FUNCTION_BLOCK Cubic_Polynomial_Interpolation
//VAR_INPUT
//	t0,t1,q0,q1,v0,v1,acc0,acc1:LREAL;	
//	t:LREAL;
//END_VAR
VAR
	h,Tp:LREAL;
	a0,a1,a2,a3:LREAL;
	targetPos,targetVel,targetAcc:LREAL;
END_VAR



//IF (t<=t1) THEN
//	pos:=a0+a1*t+a2*EXPT(t,2)+a3*EXPT(t,3);
//	vel:=a1+2*a2*t+3*a3*EXPT(t,2);
//	acc:=2*a2+6*a3*t;
//END_IF

//IF (t>t1) THEN
//	finished:=TRUE;
//	pos:=q1;
//	vel:=0;
//	acc:=0;
//ELSE
//	finished:=FALSE;
//END_IF

METHOD init : BOOL
VAR_INPUT
	t0,t1,q0,q1,v0,v1,acc0,acc1:LREAL;	
END_VAR
targetPos:=0;
targetVel:=0;
targetAcc:=0;
a0:=0;
a1:=0;
a2:=0;
a3:=0;
h:=q1-q0;
Tp:=t1-t0;

a0:=q0;
a1:=v0;
a2:=3/EXPT(Tp,2)*h-2/Tp*v0-1/Tp*v1;
a3:=-2/EXPT(Tp,3)*h+1/EXPT(Tp,2)*(v1+v0);

targetPos:=q1;
targetVel:=v1;
targetAcc:=a1;
END_METHOD

METHOD run : BOOL
VAR_INPUT
	t:LREAL;
END_VAR
VAR_IN_OUT
	pos:lreal;
	vel:lreal;
	acc:LREAL;
END_VAR
IF t>Tp THEN
	pos:=targetPos;
	vel:=targetVel;
	acc:=targetAcc;
ELSE	
	pos:=a0+a1*t+a2*EXPT(t,2)+a3*EXPT(t,3);
	vel:=a1+2*a2*t+3*a3*EXPT(t,2);
	acc:=2*a2+6*a3*t;
END_IF
END_METHOD

END_FUNCTION_BLOCK

(* stored: Version 1.1.0.1, ProductVersion 3.1.4024.12
   POU Cubic_Polynomial_Interpolation: Id {d05795ca-46ae-45d1-a565-0dbdff11dcfb}, SpecialFunc None
   Method init: Id {b4cf89e5-ebd6-4df0-a5ad-dfbeaf283d1e}
   Method run: Id {e7ad38c3-c494-4655-ac55-f8398a62ab10} *)
